# B&R Automation Studio project MappAssetInt (part 3)

#### ExportEventData.st
```iecst
// -------------------------------------------------------------------------------------------
// Read event data
// -------------------------------------------------------------------------------------------
FUNCTION_BLOCK ExportEventData
	// -------------------------------------------------------------------------------------------
	// Reset everything when enable is false
	IF NOT Enable THEN
		Status := ERR_FUB_ENABLE_FALSE;
		State := 0;
		RETURN;
	END_IF

	CASE State OF
		// -------------------------------------------------------------------------------------------
		// Wait for enable
		// -------------------------------------------------------------------------------------------
		0:
			IF Enable THEN

				// -------------------------------------------------------------------------------------------
				// Create file name
				RTC_gettime(ADR(RtcGettime));
				ExportType := ExportTypeJob;

				// Make sure we have data that can be exported
				IF RecordCount > 0 THEN
					Status := ERR_FUB_BUSY;
					CreateLoggerEntry(exASSETINT_LOG_INFO, ADR('start exporting data'), Logger);

					State := 1;
				ELSE

					CreateLoggerEntry(exASSETINT_LOG_INFO, ADR('no data to export'), Logger);
				END_IF
			END_IF

		// -------------------------------------------------------------------------------------------
		// Generate file name
		// -------------------------------------------------------------------------------------------
		1:
			// -------------------------------------------------------------------------------------------
			// Reset function blocks
			FileCreate_0.enable := FALSE;
			FileCreate_0();
			FileWrite_0.enable := FALSE;
			FileWrite_0();
			FileClose_0.enable := FALSE;
			FileClose_0();

			// -------------------------------------------------------------------------------------------
			// Export job data
			IF ExportType = ExportTypeJob THEN
				IF Configuration.JobStatistics THEN
					FileName := Configuration.JobStatisticsFileNamePattern;
				ELSE
					ExportType := ExportTypeShift;
				END_IF
			END_IF

			// -------------------------------------------------------------------------------------------
			// Export shift data
			IF ExportType = ExportTypeShift THEN
				IF Configuration.ShiftStatistics THEN
					FileName := Configuration.ShiftStatisticsFileNamePattern;
				ELSE
					ExportType := ExportTypeTimeline;
				END_IF
			END_IF

			// -------------------------------------------------------------------------------------------
			// Export timeline
			IF ExportType = ExportTypeTimeline THEN
				IF Configuration.JobStatistics THEN
					FileName := Configuration.TimelineFileNamePattern;
				ELSE
					State := 0;
					Status := ERR_OK;
					RETURN;
				END_IF
			END_IF

			// -------------------------------------------------------------------------------------------
			// Create date and time information
			ReplaceDateTime(ADR(FileName), ADR('%d'), RtcGettime.day);
			ReplaceDateTime(ADR(FileName), ADR('%m'), RtcGettime.month);
			ReplaceDateTime(ADR(FileName), ADR('%Y'), RtcGettime.year);

			ReplaceDateTime(ADR(FileName), ADR('%S'), RtcGettime.second);
			ReplaceDateTime(ADR(FileName), ADR('%M'), RtcGettime.month);
			ReplaceDateTime(ADR(FileName), ADR('%H'), RtcGettime.hour);

			idx := RecordCount - 1;
			Offset := 0;
			Status := ERR_FUB_BUSY;
			CreateLoggerEntry(exASSETINT_LOG_INFO, ADR('start exporting data'), Logger);

			State := 2;

		// -------------------------------------------------------------------------------------------
		// Delete old export file
		// -------------------------------------------------------------------------------------------
		2:
			FileDelete_0.enable := TRUE;
			FileDelete_0.pDevice := ADR(Device);
			FileDelete_0.pName := ADR(FileName);
			FileDelete_0();

			// -------------------------------------------------------------------------------------------
			// File delete successful
			IF FileDelete_0.status = ERR_OK  OR FileDelete_0.status = fiERR_FILE_NOT_FOUND THEN
				// Generate log entry
				TmpStr1 := 'delete old file ok > ';
				brsstrcat(ADR(TmpStr1), ADR(FileName));
				CreateLoggerEntry(exASSETINT_LOG_ALL, ADR(TmpStr1), Logger);

				State := 3;

			// Error
			ELSIF FileDelete_0.status <> ERR_FUB_BUSY THEN
				Status := FileDelete_0.status;
				State := 0;
			END_IF

		// -------------------------------------------------------------------------------------------
		// Create export file
		// -------------------------------------------------------------------------------------------
		3:
			FileCreate_0.enable := TRUE;
			FileCreate_0.pDevice := ADR(Device);
			FileCreate_0.pFile := ADR(FileName);
			FileCreate_0();

			// -------------------------------------------------------------------------------------------
			// File created successful
			IF FileCreate_0.status = ERR_OK THEN
				// Generate log entry
				TmpStr1 := 'create event file > ';
				brsstrcat(ADR(TmpStr1), ADR(FileName));
				CreateLoggerEntry(exASSETINT_LOG_ALL, ADR(TmpStr1), Logger);

				// Create header data depending on export file
				brsmemset(ADR(Buffer), 0, SIZEOF(Buffer));
				IF ExportType = ExportTypeJob THEN
					brsstrcat(ADR(Buffer), ADR(EXPORT_JOB_TITEL));
					brsstrcat(ADR(Buffer), ADR('$R'));
					brsstrcat(ADR(Buffer), ADR(EXPORT_JOB_HEADER));
					brsstrcat(ADR(Buffer), ADR('$R'));
				ELSIF ExportType = ExportTypeShift THEN
					brsstrcat(ADR(Buffer), ADR(EXPORT_SHIFT_TITEL));
					brsstrcat(ADR(Buffer), ADR('$R'));
					brsstrcat(ADR(Buffer), ADR(EXPORT_SHIFT_HEADER));
					brsstrcat(ADR(Buffer), ADR('$R'));
				ELSE
					brsstrcat(ADR(Buffer), ADR(EXPORT_TIMELINE_TITEL));
					brsstrcat(ADR(Buffer), ADR('$R'));
					brsstrcat(ADR(Buffer), ADR(EXPORT_TIMELINE_HEADER));
					brsstrcat(ADR(Buffer), ADR('$R'));
				END_IF

				State := 5;

			// Error
			ELSIF FileCreate_0.status <> ERR_FUB_BUSY THEN
				Status := FileCreate_0.status;
				State := 0;
			END_IF

		// -------------------------------------------------------------------------------------------
		// Generate data
		// -------------------------------------------------------------------------------------------
		4:
			// Reset buffer, copy new record
			brsmemset(ADR(Buffer), 0, SIZEOF(Buffer));
			brsmemcpy(ADR(RecordDataIntern), Memory + idx*SIZEOF(RecordDataIntern), SIZEOF(RecordDataIntern));

			// -------------------------------------------------------------------------------------------
			// Create row string for job and shift export
			IF (RecordDataIntern.EventType = RecordTypeJob AND ExportType = ExportTypeJob) OR (RecordDataIntern.EventType = RecordTypeShift AND ExportType = ExportTypeShift) THEN
				DT_TO_DTStructure(RecordDataIntern.TimeStart, ADR(DTStructure_0));
				TmpStr1 := Configuration.TimestampPattern;

				ReplaceDateTime(ADR(TmpStr1), ADR('%d'), DTStructure_0.day);
				ReplaceDateTime(ADR(TmpStr1), ADR('%m'), DTStructure_0.month);
				ReplaceDateTime(ADR(TmpStr1), ADR('%Y'), DTStructure_0.year);
				ReplaceDateTime(ADR(TmpStr1), ADR('%S'), DTStructure_0.second);
				ReplaceDateTime(ADR(TmpStr1), ADR('%M'), DTStructure_0.month);
				ReplaceDateTime(ADR(TmpStr1), ADR('%H'), DTStructure_0.hour);

				brsstrcat(ADR(Buffer), ADR(TmpStr1));
				brsstrcat(ADR(Buffer), ADR(Configuration.ColumnSeparator));

				DT_TO_DTStructure(RecordDataIntern.TimeEnd, ADR(DTStructure_0));
				TmpStr1 := Configuration.TimestampPattern;

				ReplaceDateTime(ADR(TmpStr1), ADR('%d'), DTStructure_0.day);
				ReplaceDateTime(ADR(TmpStr1), ADR('%m'), DTStructure_0.month);
				ReplaceDateTime(ADR(TmpStr1), ADR('%Y'), DTStructure_0.year);
				ReplaceDateTime(ADR(TmpStr1), ADR('%S'), DTStructure_0.second);
				ReplaceDateTime(ADR(TmpStr1), ADR('%M'), DTStructure_0.month);
				ReplaceDateTime(ADR(TmpStr1), ADR('%H'), DTStructure_0.hour);

				brsstrcat(ADR(Buffer), ADR(TmpStr1));
				brsstrcat(ADR(Buffer), ADR(Configuration.ColumnSeparator));

				brsstrcat(ADR(Buffer), ADR(RecordDataIntern.JobName));
				brsstrcat(ADR(Buffer), ADR(Configuration.ColumnSeparator));
				brsstrcat(ADR(Buffer), ADR(RecordDataIntern.CurrentUser));
				brsstrcat(ADR(Buffer), ADR(Configuration.ColumnSeparator));
				brsstrcat(ADR(Buffer), ADR(RecordDataIntern.AdditionalData));
				brsstrcat(ADR(Buffer), ADR(Configuration.ColumnSeparator));

				brsitoa(RecordDataIntern.TargetPieces, ADR(TmpStr1));
				brsstrcat(ADR(Buffer), ADR(TmpStr1));
				brsstrcat(ADR(Buffer), ADR(Configuration.ColumnSeparator));

				brsitoa(RecordDataIntern.GoodPieces, ADR(TmpStr1));
				brsstrcat(ADR(Buffer), ADR(TmpStr1));
				brsstrcat(ADR(Buffer), ADR(Configuration.ColumnSeparator));

				brsitoa(RecordDataIntern.RejectPieces, ADR(TmpStr1));
				brsstrcat(ADR(Buffer), ADR(TmpStr1));
				brsstrcat(ADR(Buffer), ADR(Configuration.ColumnSeparator));

				NormalizeFloat(RecordDataIntern.BadPieceRate, ADR(TmpStr1), Configuration);
				brsstrcat(ADR(Buffer), ADR(TmpStr1));
				brsstrcat(ADR(Buffer), ADR(Configuration.ColumnSeparator));

				lrealStr := NormalizeDateTime(RecordDataIntern.TotalTime.Hours);
				brsstrcat(ADR(Buffer), ADR(lrealStr));
				brsstrcat(ADR(Buffer), ADR(':'));
				lrealStr := NormalizeDateTime(RecordDataIntern.TotalTime.Minutes);
				brsstrcat(ADR(Buffer), ADR(lrealStr));
				brsstrcat(ADR(Buffer), ADR(':'));
				lrealStr := NormalizeDateTime(RecordDataIntern.TotalTime.Seconds);
				brsstrcat(ADR(Buffer), ADR(lrealStr));
				brsstrcat(ADR(Buffer), ADR(Configuration.ColumnSeparator));

				lrealStr := NormalizeDateTime(RecordDataIntern.ScheduledDowntime.Hours);
				brsstrcat(ADR(Buffer), ADR(lrealStr));
				brsstrcat(ADR(Buffer), ADR(':'));
				lrealStr := NormalizeDateTime(RecordDataIntern.ScheduledDowntime.Minutes);
				brsstrcat(ADR(Buffer), ADR(lrealStr));
				brsstrcat(ADR(Buffer), ADR(':'));
				lrealStr := NormalizeDateTime(RecordDataIntern.ScheduledDowntime.Seconds);
				brsstrcat(ADR(Buffer), ADR(lrealStr));
				brsstrcat(ADR(Buffer), ADR(Configuration.ColumnSeparator));

				lrealStr := NormalizeDateTime(RecordDataIntern.UnscheduledDowntime.Hours);
				brsstrcat(ADR(Buffer), ADR(lrealStr));
				brsstrcat(ADR(Buffer), ADR(':'));
				lrealStr := NormalizeDateTime(RecordDataIntern.UnscheduledDowntime.Minutes);
				brsstrcat(ADR(Buffer), ADR(lrealStr));
				brsstrcat(ADR(Buffer), ADR(':'));
				lrealStr := NormalizeDateTime(RecordDataIntern.UnscheduledDowntime.Seconds);
				brsstrcat(ADR(Buffer), ADR(lrealStr));
				brsstrcat(ADR(Buffer), ADR(Configuration.ColumnSeparator));

				lrealStr := NormalizeDateTime(RecordDataIntern.Uptime.Hours);
				brsstrcat(ADR(Buffer), ADR(lrealStr));
				brsstrcat(ADR(Buffer), ADR(':'));
				lrealStr := NormalizeDateTime(RecordDataIntern.Uptime.Minutes);
				brsstrcat(ADR(Buffer), ADR(lrealStr));
				brsstrcat(ADR(Buffer), ADR(':'));
				lrealStr := NormalizeDateTime(RecordDataIntern.Uptime.Seconds);
				brsstrcat(ADR(Buffer), ADR(lrealStr));
				brsstrcat(ADR(Buffer), ADR(Configuration.ColumnSeparator));

				lrealStr := NormalizeDateTime(RecordDataIntern.GoodProductionTime.Hours);
				brsstrcat(ADR(Buffer), ADR(lrealStr));
				brsstrcat(ADR(Buffer), ADR(':'));
				lrealStr := NormalizeDateTime(RecordDataIntern.GoodProductionTime.Minutes);
				brsstrcat(ADR(Buffer), ADR(lrealStr));
				brsstrcat(ADR(Buffer), ADR(':'));
				lrealStr := NormalizeDateTime(RecordDataIntern.GoodProductionTime.Seconds);
				brsstrcat(ADR(Buffer), ADR(lrealStr));
				brsstrcat(ADR(Buffer), ADR(Configuration.ColumnSeparator));

				lrealStr := NormalizeDateTime(RecordDataIntern.NominalProductionTime.Hours);
				brsstrcat(ADR(Buffer), ADR(lrealStr));
				brsstrcat(ADR(Buffer), ADR(':'));
				lrealStr := NormalizeDateTime(RecordDataIntern.NominalProductionTime.Minutes);
				brsstrcat(ADR(Buffer), ADR(lrealStr));
				brsstrcat(ADR(Buffer), ADR(':'));
				lrealStr := NormalizeDateTime(RecordDataIntern.NominalProductionTime.Seconds);
				brsstrcat(ADR(Buffer), ADR(lrealStr));
				brsstrcat(ADR(Buffer), ADR(Configuration.ColumnSeparator));

				NormalizeFloat(RecordDataIntern.NominalProductionTimeRate, ADR(TmpStr1), Configuration);
				brsstrcat(ADR(Buffer), ADR(TmpStr1));
				brsstrcat(ADR(Buffer), ADR(Configuration.ColumnSeparator));

				NormalizeFloat(RecordDataIntern.ScheduledDowntimeRate, ADR(TmpStr1), Configuration);
				brsstrcat(ADR(Buffer), ADR(TmpStr1));
				brsstrcat(ADR(Buffer), ADR(Configuration.ColumnSeparator));

				NormalizeFloat(RecordDataIntern.UnscheduledDowntimeRate, ADR(TmpStr1), Configuration);
				brsstrcat(ADR(Buffer), ADR(TmpStr1));
				brsstrcat(ADR(Buffer), ADR(Configuration.ColumnSeparator));

				NormalizeFloat(RecordDataIntern.CurrentProductionRate, ADR(TmpStr1), Configuration);
				brsstrcat(ADR(Buffer), ADR(TmpStr1));
				brsstrcat(ADR(Buffer), ADR(Configuration.ColumnSeparator));

				brsstrcat(ADR(Buffer), ADR(RecordDataIntern.ShiftName));
				brsstrcat(ADR(Buffer), ADR(Configuration.ColumnSeparator));
				brsstrcat(ADR(Buffer), ADR('$R'));

				State := 5;
			END_IF

			// -------------------------------------------------------------------------------------------
			// Export data for timeline

			IF (RecordDataIntern.EventType >= RecordTypeNoShift AND ExportType = ExportTypeTimeline) THEN
				// Create start time
				DT_TO_DTStructure(RecordDataIntern.TimeStart, ADR(DTStructure_0));
				TmpStr1 := Configuration.TimestampPattern;

				ReplaceDateTime(ADR(TmpStr1), ADR('%d'), DTStructure_0.day);
				ReplaceDateTime(ADR(TmpStr1), ADR('%m'), DTStructure_0.month);
				ReplaceDateTime(ADR(TmpStr1), ADR('%Y'), DTStructure_0.year);
				ReplaceDateTime(ADR(TmpStr1), ADR('%S'), DTStructure_0.second);
				ReplaceDateTime(ADR(TmpStr1), ADR('%M'), DTStructure_0.month);
				ReplaceDateTime(ADR(TmpStr1), ADR('%H'), DTStructure_0.hour);

				brsstrcat(ADR(Buffer), ADR(TmpStr1));
				brsstrcat(ADR(Buffer), ADR(Configuration.ColumnSeparator));

				// Add shift name
				brsstrcat(ADR(Buffer), ADR(RecordDataIntern.ShiftName));
				brsstrcat(ADR(Buffer), ADR(Configuration.ColumnSeparator));

				// Event is scheduled downtime
				IF RecordDataIntern.EventType = RecordTypeNoShift THEN
					brsstrcat(ADR(Buffer), ADR('No shift'));
				// Event is scheduled downtime
				ELSIF RecordDataIntern.EventType = RecordTypeDowntimeScheduled THEN
					brsstrcat(ADR(Buffer), ADR('Scheduled Downtime'));
				// Event is unscheduled downtime
				ELSIF RecordDataIntern.EventType = RecordTypeDowntimeUnscheduled THEN
					brsstrcat(ADR(Buffer), ADR('Unscheduled Downtime'));
				// Event is new shift
				ELSE
					brsstrcat(ADR(Buffer), ADR('Uptime'));
				END_IF
				brsstrcat(ADR(Buffer), ADR(Configuration.ColumnSeparator));

				// Additional data
				brsstrcat(ADR(Buffer), ADR(RecordDataIntern.AdditionalData));
				brsstrcat(ADR(Buffer), ADR(Configuration.ColumnSeparator));

				// Total time
				lrealStr := NormalizeDateTime(RecordDataIntern.TotalTime.Hours);
				brsstrcat(ADR(Buffer), ADR(lrealStr));
				brsstrcat(ADR(Buffer), ADR(':'));
				lrealStr := NormalizeDateTime(RecordDataIntern.TotalTime.Minutes);
				brsstrcat(ADR(Buffer), ADR(lrealStr));
				brsstrcat(ADR(Buffer), ADR(':'));
				lrealStr := NormalizeDateTime(RecordDataIntern.TotalTime.Seconds);
				brsstrcat(ADR(Buffer), ADR(lrealStr));
				brsstrcat(ADR(Buffer), ADR(Configuration.ColumnSeparator));

				// Job name
				brsstrcat(ADR(Buffer), ADR(RecordDataIntern.JobName));
				brsstrcat(ADR(Buffer), ADR(Configuration.ColumnSeparator));

				brsstrcat(ADR(Buffer), ADR('$R'));

				State := 5;
			END_IF

			// Increase counter
			IF idx = 0 THEN
				State := 6;
			ELSE
				idx := idx - 1;
			END_IF

		// -------------------------------------------------------------------------------------------
		// Write data
		// -------------------------------------------------------------------------------------------
		5:
			FileWrite_0.enable := TRUE;
			FileWrite_0.ident := FileCreate_0.ident;
			FileWrite_0.offset := Offset;
			FileWrite_0.pSrc := ADR(Buffer);
			FileWrite_0.len := brsstrlen(ADR(Buffer));
			FileWrite_0();

			// File created successful
			IF FileWrite_0.status = ERR_OK THEN
				// Generate log entry
				TmpStr1 := 'write idx ok > ';
				brsitoa(idx, ADR(TmpStr2));
				brsstrcat(ADR(TmpStr1), ADR(TmpStr2));
				CreateLoggerEntry(exASSETINT_LOG_ALL, ADR(TmpStr1), Logger);

				// Remember offset
				Offset := Offset + FileWrite_0.len;

				// Go to next step
				IF idx > 0 THEN
					State := 4;
				ELSE
					State := 6;
				END_IF

				// Error
			ELSIF FileWrite_0.status <> ERR_FUB_BUSY THEN
				Status := FileWrite_0.status;
				State := 0;
			END_IF

			// -------------------------------------------------------------------------------------------
			// Close file
			// -------------------------------------------------------------------------------------------
		6:
			FileClose_0.enable := TRUE;
			FileClose_0.ident := FileCreate_0.ident;
			FileClose_0();

			// File created successful
			IF FileClose_0.status = ERR_OK THEN
				// Generate log entry
				TmpStr1 := 'close export file ok > ';
				brsstrcat(ADR(TmpStr1), ADR(FileName));
				CreateLoggerEntry(exASSETINT_LOG_ALL, ADR(TmpStr1), Logger);

				// Proceed with shift export
				IF ExportType = ExportTypeJob THEN
					ExportType := ExportTypeShift;
					State := 1;
					// Proceed with timeline export
				ELSIF ExportType = ExportTypeShift THEN
					ExportType := ExportTypeTimeline;
					State := 1;
				ELSE
					// Finish up
					Status := ERR_OK;
					State := 0;
				END_IF

				// Error
			ELSIF FileClose_0.status <> ERR_FUB_BUSY THEN
				Status := FileClose_0.status;
				State := 0;
			END_IF
	END_CASE;

END_FUNCTION_BLOCK

// -------------------------------------------------------------------------------------------
// Format float according to configuration
// -------------------------------------------------------------------------------------------
FUNCTION NormalizeFloat
	brsftoa(value, ADR(tmpStr));
	idx := FindInstr(ADR(tmpStr), ADR('.')) + configuration.DecimalDigits + 1;
	IF idx >= brsstrlen(ADR(tmpStr)) THEN
		brsstrcpy(output, ADR(tmpStr));
	ELSE
		brsmemcpy(output, ADR(tmpStr), idx);
		brsmemset(output + idx, 0, 1);
	END_IF
	ReplaceString(output, ADR('.'), ADR(configuration.DecimalMark));
END_FUNCTION

// -------------------------------------------------------------------------------------------
// Add additional 0 when value is < 10
// -------------------------------------------------------------------------------------------
FUNCTION NormalizeDateTime
	IF(value < 10) THEN
		TmpStr1 := '0';
	ELSE
		TmpStr1 := '';
	END_IF
	brsitoa(value, ADR(TmpStr2));
	brsstrcat(ADR(TmpStr1), ADR(TmpStr2));

	brsmemcpy(ADR(NormalizeDateTime), ADR(TmpStr1), brsstrlen(ADR(TmpStr1)));

END_FUNCTION

// -------------------------------------------------------------------------------------------
// Find and replace date and time information
// -------------------------------------------------------------------------------------------
FUNCTION ReplaceDateTime
	lrealStr := NormalizeDateTime(value);
	ReplaceString(dataSTR, searchSTR, ADR(lrealStr));

	ReplaceDateTime := TRUE;
END_FUNCTION

// -------------------------------------------------------------------------------------------
// Find and replace string
// -------------------------------------------------------------------------------------------
FUNCTION ReplaceString
	IF (brsstrlen(dataSTR) >= brsstrlen(searchSTR)) THEN
		FOR idx:=0 TO brsstrlen(dataSTR) - brsstrlen(searchSTR) DO
			IF (brsmemcmp(dataSTR + idx, searchSTR, brsstrlen(searchSTR)) = 0) THEN
				// Move data around
				brsmemmove(dataSTR + idx + brsstrlen(replaceSTR), dataSTR + idx + brsstrlen(searchSTR), brsstrlen(dataSTR) - brsstrlen(searchSTR) + 1);
				brsmemcpy(dataSTR + idx, replaceSTR, brsstrlen(replaceSTR));
				// Set found flag and exit if only one hit is needed
				ReplaceString := TRUE;
				// Correct index for next search
				IF(brsstrlen(replaceSTR) > 0) THEN
					idx := idx + brsstrlen(replaceSTR);
				END_IF
				idx := idx - 1;
				// Exit if no data is left
				IF (brsstrlen(dataSTR) = 0 OR brsstrlen(dataSTR) < brsstrlen(searchSTR)) THEN
					EXIT;
				END_IF
			END_IF
		END_FOR;
	END_IF
END_FUNCTION
```

#### WriteConfiguration.st
```iecst
// -------------------------------------------------------------------------------------------
// Write configuration
// -------------------------------------------------------------------------------------------
FUNCTION_BLOCK WriteConfiguration
	// -------------------------------------------------------------------------------------------
	// Reset everything when enable is false
	IF NOT Enable THEN
		Status := ERR_FUB_ENABLE_FALSE;
		State := 0;
		RETURN;
	END_IF

	CASE State OF
		// -------------------------------------------------------------------------------------------
		// Wait for enable
		0:
			IF Enable THEN
				// Reset function blocks
				FileOpen_0.enable := FALSE;
				FileOpen_0();
				FileCreate_0.enable := FALSE;
				FileCreate_0();
				FileWrite_0.enable := FALSE;
				FileWrite_0();
				FileClose_0.enable := FALSE;
				FileClose_0();

				Status := ERR_FUB_BUSY;
				CreateLoggerEntry(exASSETINT_LOG_INFO, ADR('save configuration'), Logger);
				State := 1;
			END_IF

			// -------------------------------------------------------------------------------------------
			// Open file
		1:
			FileOpen_0.enable := TRUE;
			FileOpen_0.pDevice := ADR(Device);
			FileOpen_0.pFile := ADR('exAssetConfig');
			FileOpen_0.mode := fiREAD_WRITE;
			FileOpen_0();

			// File opened successful
			IF FileOpen_0.status = ERR_OK THEN
				// Generate log entry
				CreateLoggerEntry(exASSETINT_LOG_ALL, ADR('open configuration file ok'), Logger);

				// Remember ident go to next step
				Ident := FileOpen_0.ident;
				State := 3;

			// Create event file when it does not exist
			ELSIF FileOpen_0.status = fiERR_FILE_NOT_FOUND  THEN
				State := 2;

			// Error
			ELSIF FileOpen_0.status <> ERR_FUB_BUSY THEN
				Status := FileOpen_0.status;
				State := 0;
			END_IF

			// -------------------------------------------------------------------------------------------
			// Create file
		2:
			FileCreate_0.enable := TRUE;
			FileCreate_0.pDevice := ADR(Device);
			FileCreate_0.pFile := ADR('exAssetConfig');
			FileCreate_0();

			// File created successful
			IF FileCreate_0.status = ERR_OK THEN
				// Generate log entry
				CreateLoggerEntry(exASSETINT_LOG_ALL, ADR('created configuration file'), Logger);

				// Remember ident go to next step
				Ident := FileCreate_0.ident;
				State := 3;

				// Error
			ELSIF FileCreate_0.status <> ERR_FUB_BUSY THEN
				Status := FileCreate_0.status;
				State := 0;
			END_IF

			// -------------------------------------------------------------------------------------------
			// Write data
		3:
			FileWrite_0.enable := TRUE;
			FileWrite_0.ident := Ident;
			FileWrite_0.pSrc := ADR(Configuration);
			FileWrite_0.len := SIZEOF(Configuration);
			FileWrite_0();

			// File created successful
			IF FileWrite_0.status = ERR_OK THEN
				// Generate log entry
				CreateLoggerEntry(exASSETINT_LOG_ALL, ADR('write configuration file ok'), Logger);

				// Go to next step
				State := 4;

			// Error
			ELSIF FileWrite_0.status <> ERR_FUB_BUSY THEN
				Status := FileWrite_0.status;
				State := 0;
			END_IF

			// -------------------------------------------------------------------------------------------
			// Close file
		4:
			FileClose_0.enable := TRUE;
			FileClose_0.ident := Ident;
			FileClose_0();

			// File created successful
			IF FileClose_0.status = ERR_OK THEN
				// Generate log entry
				CreateLoggerEntry(exASSETINT_LOG_ALL, ADR('close configuration file ok'), Logger);

				// Finish up
				Status := ERR_OK;
				State := 0;

				// Error
			ELSIF FileClose_0.status <> ERR_FUB_BUSY THEN
				Status := FileClose_0.status;
				State := 0;
			END_IF
	END_CASE;

END_FUNCTION_BLOCK
```

#### ReadConfiguration.st
```iecst
// -------------------------------------------------------------------------------------------
// Read configuration
// -------------------------------------------------------------------------------------------
FUNCTION_BLOCK ReadConfiguration
	// -------------------------------------------------------------------------------------------
	// Reset everything when enable is false
	IF NOT Enable THEN
		Status := ERR_FUB_ENABLE_FALSE;
		State := 0;
		RETURN;
	END_IF

	CASE State OF
		// -------------------------------------------------------------------------------------------
		// Wait for enable
		0:
			IF Enable THEN
				// Reset function blocks
				FileOpen_0.enable := FALSE;
				FileOpen_0();
				FileRead_0.enable := FALSE;
				FileRead_0();
				FileClose_0.enable := FALSE;
				FileClose_0();

				Status := ERR_FUB_BUSY;
				CreateLoggerEntry(exASSETINT_LOG_INFO, ADR('reading configuration'), Logger);
				State := 1;
			END_IF

		// -------------------------------------------------------------------------------------------
		// Open event file
		1:
			// Open file
			FileOpen_0.enable := TRUE;
			FileOpen_0.pDevice := ADR(Device);
			FileOpen_0.pFile := ADR('exAssetConfig');
			FileOpen_0.mode := fiREAD_ONLY;
			FileOpen_0();

			// File opened successful
			IF FileOpen_0.status = ERR_OK THEN
				// Generate log entry
				CreateLoggerEntry(exASSETINT_LOG_ALL, ADR('opened event configuration'), Logger);

				// Go to next step
				State := 5;

			// Error
			ELSIF FileOpen_0.status <> ERR_FUB_BUSY THEN
				Status := FileOpen_0.status;
				State := 0;
			END_IF

		// -------------------------------------------------------------------------------------------
		// Read configuration data
		5:
			FileRead_0.enable := TRUE;
			FileRead_0.ident := FileOpen_0.ident;
			FileRead_0.pDest := ADR(Configuration);
			FileRead_0.len := FileOpen_0.filelen;
			FileRead_0();

			// File read successful
			IF FileRead_0.status = ERR_OK THEN
				// Generate log entry
				CreateLoggerEntry(exASSETINT_LOG_ALL, ADR('read event configuration'), Logger);

				State := 6;

			// Error
			ELSIF FileRead_0.status <> ERR_FUB_BUSY THEN
				Status := FileRead_0.status;
				State := 0;
			END_IF

		// -------------------------------------------------------------------------------------------
		// Close file
		6:
			FileClose_0.enable := TRUE;
			FileClose_0.ident := FileOpen_0.ident;
			FileClose_0();

			// File closed successful
			IF FileClose_0.status = ERR_OK THEN
				// Generate log entry
				CreateLoggerEntry(exASSETINT_LOG_ALL, ADR('closed event configuration'), Logger);

				// Go to next step
				Status := ERR_OK;
				State := 0;

				// Error
			ELSIF FileClose_0.status <> ERR_FUB_BUSY THEN
				Status := FileClose_0.status;
				State := 0;
			END_IF
	END_CASE;

END_FUNCTION_BLOCK
```

#### ReadLinkData.st
```iecst
// -------------------------------------------------------------------------------------------
// File version 1001
// -------------------------------------------------------------------------------------------
// Read configuration
// -------------------------------------------------------------------------------------------
FUNCTION_BLOCK ReadLinkData
	// -------------------------------------------------------------------------------------------
	// Reset everything when enable is false
	IF NOT Enable THEN
		Status := ERR_FUB_ENABLE_FALSE;
		State := 0;
		RETURN;
	END_IF

	CASE State OF
		// -------------------------------------------------------------------------------------------
		// Wait for enable
		0:
			IF Enable THEN
				// Reset function blocks
				FileOpen_0.enable := FALSE;
				FileOpen_0();
				FileRead_0.enable := FALSE;
				FileRead_0();
				FileClose_0.enable := FALSE;
				FileClose_0();

				Status := ERR_FUB_BUSY;
				CreateLoggerEntry(exASSETINT_LOG_INFO, ADR('reading link data'), Logger);
				State := 1;
			END_IF

		// -------------------------------------------------------------------------------------------
		// Open event file
		1:
			// Open file
			FileOpen_0.enable := TRUE;
			FileOpen_0.pDevice := ADR(Device);
			FileOpen_0.pFile := ADR('exAssetLink');
			FileOpen_0.mode := fiREAD_ONLY;
			FileOpen_0();

			// File opened successful
			IF FileOpen_0.status = ERR_OK THEN
				// Make sure backup data has correct size
				IF FileOpen_0.filelen <> SIZEOF(LinkRead) THEN
					CreateLoggerEntry(exASSETINT_LOG_ERROR, ADR('link backup data size is incorrect'), Logger);
					StatusRead := ERR_ASSET_LINK_SIZE;

					State := 6;
				ELSE
					CreateLoggerEntry(exASSETINT_LOG_ALL, ADR('open link data ok'), Logger);
					State := 5;
				END_IF

				// Error
			ELSIF FileOpen_0.status <> ERR_FUB_BUSY THEN
				Status := FileOpen_0.status;
				State := 0;
			END_IF

		// -------------------------------------------------------------------------------------------
		// Read configuration data
		5:
			FileRead_0.enable := TRUE;
			FileRead_0.ident := FileOpen_0.ident;
			FileRead_0.pDest := ADR(LinkRead);
			FileRead_0.len := FileOpen_0.filelen;
			FileRead_0();

			// File read successful
			IF FileRead_0.status = ERR_OK THEN
				// Make sure backup version is correct
				IF LinkRead.Version <> EXLINK_VERSION THEN
					CreateLoggerEntry(exASSETINT_LOG_ERROR, ADR('link backup data version is incorrect'), Logger);
					StatusRead := ERR_ASSET_LINK_VERSION;

				ELSE
					brsmemcpy(ADR(Link), ADR(LinkRead), SIZEOF(LinkRead));
					CreateLoggerEntry(exASSETINT_LOG_ALL, ADR('open link data ok'), Logger);
				END_IF

				State := 6;

			// Error
			ELSIF FileRead_0.status <> ERR_FUB_BUSY THEN
				Status := FileRead_0.status;
				State := 0;
			END_IF

		// -------------------------------------------------------------------------------------------
		// Close file
		6:
			FileClose_0.enable := TRUE;
			FileClose_0.ident := FileOpen_0.ident;
			FileClose_0();

			// File closed successful
			IF FileClose_0.status = ERR_OK THEN
				// Auto delete corrupt file
				IF StatusRead <> 0 THEN
					State := 7;
				ELSE
					// Generate log entry
					CreateLoggerEntry(exASSETINT_LOG_ALL, ADR('closed link data ok'), Logger);

					// Go to next step
					Status := ERR_OK;
					State := 0;
				END_IF

			// Error
			ELSIF FileClose_0.status <> ERR_FUB_BUSY THEN
				Status := FileClose_0.status;
				State := 0;
			END_IF

			// -------------------------------------------------------------------------------------------
			// Delete corrupt file
		7:
			FileDelete_0.enable := TRUE;
			FileDelete_0.pDevice := ADR(Device);
			FileDelete_0.pName := ADR('exAssetLink');
			FileDelete_0();

			// File delete successful
			IF FileDelete_0.status = ERR_OK THEN
				// Generate log entry
				CreateLoggerEntry(exASSETINT_LOG_ALL, ADR('delete corrupt link backup file ok'), Logger);

				Status := StatusRead;
				State := 0;

				// Error
			ELSIF FileDelete_0.status <> ERR_FUB_BUSY THEN
				Status := FileDelete_0.status;
				State := 0;
			END_IF
	END_CASE;

END_FUNCTION_BLOCK
```

#### WriteLinkData.st
```iecst
// -------------------------------------------------------------------------------------------
// File version 1000
// -------------------------------------------------------------------------------------------
// Write configuration
// -------------------------------------------------------------------------------------------
FUNCTION_BLOCK WriteLinkData
	// -------------------------------------------------------------------------------------------
	// Reset everything when enable is false
	IF NOT Enable THEN
		Status := ERR_FUB_ENABLE_FALSE;
		State := 0;
		RETURN;
	END_IF

	CASE State OF
		// -------------------------------------------------------------------------------------------
		// Wait for enable
		0:
			IF Enable THEN
				// Reset function blocks
				FileOpen_0.enable := FALSE;
				FileOpen_0();
				FileCreate_0.enable := FALSE;
				FileCreate_0();
				FileWrite_0.enable := FALSE;
				FileWrite_0();
				FileClose_0.enable := FALSE;
				FileClose_0();

				Status := ERR_FUB_BUSY;
				CreateLoggerEntry(exASSETINT_LOG_INFO, ADR('saving link data'), Logger);
				State := 1;
			END_IF

			// -------------------------------------------------------------------------------------------
			// Open file
		1:
			FileOpen_0.enable := TRUE;
			FileOpen_0.pDevice := ADR(Device);
			FileOpen_0.pFile := ADR('exAssetLink');
			FileOpen_0.mode := fiREAD_WRITE;
			FileOpen_0();

			// File opened successful
			IF FileOpen_0.status = ERR_OK THEN
				// Generate log entry
				CreateLoggerEntry(exASSETINT_LOG_ALL, ADR('open link data ok'), Logger);

				// Remember ident go to next step
				Ident := FileOpen_0.ident;
				State := 3;

			// Create event file when it does not exist
			ELSIF FileOpen_0.status = fiERR_FILE_NOT_FOUND  THEN
				State := 2;

			// Error
			ELSIF FileOpen_0.status <> ERR_FUB_BUSY THEN
				Status := FileOpen_0.status;
				State := 0;
			END_IF

			// -------------------------------------------------------------------------------------------
			// Create file
		2:
			FileCreate_0.enable := TRUE;
			FileCreate_0.pDevice := ADR(Device);
			FileCreate_0.pFile := ADR('exAssetLink');
			FileCreate_0();

			// File created successful
			IF FileCreate_0.status = ERR_OK THEN
				// Generate log entry
				CreateLoggerEntry(exASSETINT_LOG_ALL, ADR('create link data file'), Logger);

				// Remember ident go to next step
				Ident := FileCreate_0.ident;
				State := 3;

				// Error
			ELSIF FileCreate_0.status <> ERR_FUB_BUSY THEN
				Status := FileCreate_0.status;
				State := 0;
			END_IF

			// -------------------------------------------------------------------------------------------
			// Write data
		3:
			FileWrite_0.enable := TRUE;
			FileWrite_0.ident := Ident;
			FileWrite_0.pSrc := ADR(Link);
			FileWrite_0.len := SIZEOF(Link);
			FileWrite_0();

			// File created successful
			IF FileWrite_0.status = ERR_OK THEN
				// Generate log entry
				CreateLoggerEntry(exASSETINT_LOG_ALL, ADR('write link data ok'), Logger);

				// Go to next step
				State := 4;

			// Error
			ELSIF FileWrite_0.status <> ERR_FUB_BUSY THEN
				Status := FileWrite_0.status;
				State := 0;
			END_IF

			// -------------------------------------------------------------------------------------------
			// Close file
		4:
			FileClose_0.enable := TRUE;
			FileClose_0.ident := Ident;
			FileClose_0();

			// File created successful
			IF FileClose_0.status = ERR_OK THEN
				// Generate log entry
				CreateLoggerEntry(exASSETINT_LOG_ALL, ADR('close link data ok'), Logger);

				// Finish up
				Status := ERR_OK;
				State := 0;

				// Error
			ELSIF FileClose_0.status <> ERR_FUB_BUSY THEN
				Status := FileClose_0.status;
				State := 0;
			END_IF
	END_CASE;

END_FUNCTION_BLOCK
```

#### CalcStats.st
```iecst
// -------------------------------------------------------------------------------------------
// File version 1002
// -------------------------------------------------------------------------------------------
// Calculate current job statistics
FUNCTION CalcStatsJob
	// -------------------------------------------------------------------------------------------
	// Calculate total time, remember total time in milliseconds for accuaracy but convert to seconds for local calculations
	exLink.JobTotalTime := exLink.JobTotalTime + DiffLastCall;
	JobTotalTime := LREAL_TO_UDINT(exLink.JobTotalTime/1000);

	exLink.JobStatistics.TotalTime.Hours := JobTotalTime/3600;
	exLink.JobStatistics.TotalTime.Minutes := UDINT_TO_USINT((JobTotalTime - exLink.JobStatistics.TotalTime.Hours*3600)/60);
	exLink.JobStatistics.TotalTime.Seconds := UDINT_TO_USINT(JobTotalTime - exLink.JobStatistics.TotalTime.Hours*3600 - exLink.JobStatistics.TotalTime.Minutes*60);

	// Calculate scheduled downtime
	IF Downtime = exASSETINT_SCHEDULED_DOWNTIME THEN
		exLink.JobDowntimeScheduled := exLink.JobDowntimeScheduled + DiffLastCall;
		exLink.JobStatistics.ScheduledDowntime.Hours := exLink.JobDowntimeScheduled/3600000;
		exLink.JobStatistics.ScheduledDowntime.Minutes := UDINT_TO_USINT((exLink.JobDowntimeScheduled - exLink.JobStatistics.ScheduledDowntime.Hours*3600000)/60000);
		exLink.JobStatistics.ScheduledDowntime.Seconds := UDINT_TO_USINT((exLink.JobDowntimeScheduled - exLink.JobStatistics.ScheduledDowntime.Hours*3600000 - exLink.JobStatistics.ScheduledDowntime.Minutes*60000)/1000);
	END_IF

	// Calculate unscheduled downtime
	IF Downtime = exASSETINT_UNSCHEDULED_DOWNTIME THEN
		exLink.JobDowntimeUnscheduled := exLink.JobDowntimeUnscheduled + DiffLastCall;
		exLink.JobStatistics.UnscheduledDowntime.Hours := exLink.JobDowntimeUnscheduled/3600000;
		exLink.JobStatistics.UnscheduledDowntime.Minutes := UDINT_TO_USINT((exLink.JobDowntimeUnscheduled - exLink.JobStatistics.UnscheduledDowntime.Hours*3600000)/60000);
		exLink.JobStatistics.UnscheduledDowntime.Seconds := UDINT_TO_USINT((exLink.JobDowntimeUnscheduled - exLink.JobStatistics.UnscheduledDowntime.Hours*3600000 - exLink.JobStatistics.UnscheduledDowntime.Minutes*60000)/1000);
	END_IF

	// Calculate uptime
	IF Downtime = exASSETINT_NO_DOWNTIME THEN
		Uptime := JobTotalTime - exLink.JobDowntimeScheduled/1000 - exLink.JobDowntimeUnscheduled/1000;
		exLink.JobStatistics.Uptime.Hours := Uptime/3600;
		exLink.JobStatistics.Uptime.Minutes := UDINT_TO_USINT((Uptime - exLink.JobStatistics.Uptime.Hours*3600)/60);
		exLink.JobStatistics.Uptime.Seconds := UDINT_TO_USINT(Uptime - exLink.JobStatistics.Uptime.Hours*3600 - exLink.JobStatistics.Uptime.Minutes*60);
	END_IF

	// -------------------------------------------------------------------------------------------
	// Calculate counters
	IF exLink.JobStatistics.TotalPieces > exLink.JobStatistics.RejectPieces THEN
		exLink.JobStatistics.GoodPieces := exLink.JobStatistics.TotalPieces - exLink.JobStatistics.RejectPieces;
	ELSE
		exLink.JobStatistics.GoodPieces := 0;
		exLink.JobStatistics.RejectPieces := exLink.JobStatistics.TotalPieces;
	END_IF
	IF exLink.JobStatistics.TotalPieces > 0 THEN
		exLink.JobStatistics.BadPieceRate := UDINT_TO_REAL(exLink.JobStatistics.RejectPieces)/UDINT_TO_REAL(exLink.JobStatistics.TotalPieces);
	END_IF

	// -------------------------------------------------------------------------------------------
	// Additional times and rates
	NominalProductionTime := REAL_TO_UDINT(UDINT_TO_REAL(exLink.JobStatistics.TotalPieces)*(3600/Parameter.NominalProductionRate));
	exLink.JobStatistics.NominalProductionTime.Hours := NominalProductionTime/3600;
	exLink.JobStatistics.NominalProductionTime.Minutes := UDINT_TO_USINT((NominalProductionTime - exLink.JobStatistics.NominalProductionTime.Hours*3600)/60);
	exLink.JobStatistics.NominalProductionTime.Seconds := UDINT_TO_USINT(NominalProductionTime - exLink.JobStatistics.NominalProductionTime.Hours*3600 - exLink.JobStatistics.NominalProductionTime.Minutes*60);

	GoodProductionTime := REAL_TO_UDINT(UDINT_TO_REAL(exLink.JobStatistics.GoodPieces)*(3600/Parameter.NominalProductionRate));
	exLink.JobStatistics.GoodProductionTime.Hours := GoodProductionTime/3600;
	exLink.JobStatistics.GoodProductionTime.Minutes := UDINT_TO_USINT((GoodProductionTime - exLink.JobStatistics.GoodProductionTime.Hours*3600)/60);
	exLink.JobStatistics.GoodProductionTime.Seconds := UDINT_TO_USINT(GoodProductionTime - exLink.JobStatistics.GoodProductionTime.Hours*3600 - exLink.JobStatistics.GoodProductionTime.Minutes*60);

	IF exLink.JobDowntimeScheduled > 0 AND JobTotalTime > 0 THEN
		exLink.JobStatistics.ScheduledDowntimeRate := UDINT_TO_REAL(exLink.JobDowntimeScheduled/JobTotalTime)/1000;
	END_IF
	IF exLink.JobDowntimeUnscheduled > 0 AND JobTotalTime > 0 THEN
		exLink.JobStatistics.UnscheduledDowntimeRate := UDINT_TO_REAL(exLink.JobDowntimeUnscheduled/JobTotalTime)/1000;
	END_IF
	IF Uptime > 0 THEN
		exLink.JobStatistics.NominalProductionTimeRate := UDINT_TO_REAL(NominalProductionTime)/UDINT_TO_REAL(Uptime);
	END_IF
	IF JobTotalTime > 0 THEN
		exLink.JobStatistics.CurrentProductionRate := UDINT_TO_REAL(exLink.JobStatistics.TotalPieces)/UDINT_TO_REAL(JobTotalTime)*3600;
	END_IF

	brsmemcpy(ADR(JobStatistics), ADR(exLink.JobStatistics), SIZEOF(exLink.JobStatistics));
	CalcStatsJob := TRUE;
END_FUNCTION

// -------------------------------------------------------------------------------------------
// Calculate current shift statistics
FUNCTION CalcStatsShift
	// -------------------------------------------------------------------------------------------
	// Calculate total time, remember total time in milliseconds for accuaracy but convert to seconds for local calculations
	exLink.ShiftTotalTime := exLink.ShiftTotalTime + DiffLastCall;
	ShiftTotalTime := LREAL_TO_UDINT(exLink.ShiftTotalTime/1000);

	exLink.ShiftStatistics.TotalTime.Hours := ShiftTotalTime/3600;
	exLink.ShiftStatistics.TotalTime.Minutes := UDINT_TO_USINT((ShiftTotalTime - exLink.ShiftStatistics.TotalTime.Hours*3600)/60);
	exLink.ShiftStatistics.TotalTime.Seconds := UDINT_TO_USINT(ShiftTotalTime - exLink.ShiftStatistics.TotalTime.Hours*3600 - exLink.ShiftStatistics.TotalTime.Minutes*60);

	// Calculate scheduled downtime
	IF Downtime = exASSETINT_SCHEDULED_DOWNTIME THEN
		exLink.ShiftDowntimeScheduled := exLink.ShiftDowntimeScheduled + DiffLastCall;
		exLink.ShiftStatistics.ScheduledDowntime.Hours := exLink.ShiftDowntimeScheduled/3600000;
		exLink.ShiftStatistics.ScheduledDowntime.Minutes := UDINT_TO_USINT((exLink.ShiftDowntimeScheduled - exLink.ShiftStatistics.ScheduledDowntime.Hours*3600000)/60000);
		exLink.ShiftStatistics.ScheduledDowntime.Seconds := UDINT_TO_USINT((exLink.ShiftDowntimeScheduled - exLink.ShiftStatistics.ScheduledDowntime.Hours*3600000 - exLink.ShiftStatistics.ScheduledDowntime.Minutes*60000)/1000);
	END_IF

	// Calculate scheduled downtime
	IF Downtime = exASSETINT_UNSCHEDULED_DOWNTIME THEN
		exLink.ShiftDowntimeUnscheduled := exLink.ShiftDowntimeUnscheduled + DiffLastCall;
		exLink.ShiftStatistics.UnscheduledDowntime.Hours := exLink.ShiftDowntimeUnscheduled/3600000;
		exLink.ShiftStatistics.UnscheduledDowntime.Minutes := UDINT_TO_USINT((exLink.ShiftDowntimeUnscheduled - exLink.ShiftStatistics.UnscheduledDowntime.Hours*3600000)/60000);
		exLink.ShiftStatistics.UnscheduledDowntime.Seconds := UDINT_TO_USINT((exLink.ShiftDowntimeUnscheduled - exLink.ShiftStatistics.UnscheduledDowntime.Hours*3600000 - exLink.ShiftStatistics.UnscheduledDowntime.Minutes*60000)/1000);
	END_IF

	// Calculate uptime
	IF Downtime = exASSETINT_NO_DOWNTIME THEN
		Uptime := ShiftTotalTime - exLink.ShiftDowntimeScheduled/1000 - exLink.ShiftDowntimeUnscheduled/1000;
		exLink.ShiftStatistics.Uptime.Hours := Uptime/3600;
		exLink.ShiftStatistics.Uptime.Minutes := UDINT_TO_USINT((Uptime - exLink.ShiftStatistics.Uptime.Hours*3600)/60);
		exLink.ShiftStatistics.Uptime.Seconds := UDINT_TO_USINT(Uptime - exLink.ShiftStatistics.Uptime.Hours*3600 - exLink.ShiftStatistics.Uptime.Minutes*60);
	END_IF

	// -------------------------------------------------------------------------------------------
	// Calculate counters
	exLink.ShiftStatistics.TargetPieces := LREAL_TO_UDINT(UDINT_TO_REAL(ShiftTotalTime)/3600*Parameter.NominalProductionRate);
	IF exLink.ShiftStatistics.TotalPieces > exLink.ShiftStatistics.RejectPieces THEN
		exLink.ShiftStatistics.GoodPieces := exLink.ShiftStatistics.TotalPieces - exLink.ShiftStatistics.RejectPieces;
	ELSE
		exLink.ShiftStatistics.GoodPieces := 0;
		exLink.ShiftStatistics.RejectPieces := exLink.ShiftStatistics.TotalPieces;
	END_IF
	IF exLink.ShiftStatistics.TotalPieces > 0 THEN
		exLink.ShiftStatistics.BadPieceRate := UDINT_TO_REAL(exLink.ShiftStatistics.RejectPieces)/UDINT_TO_REAL(exLink.ShiftStatistics.TotalPieces);
	END_IF

	// -------------------------------------------------------------------------------------------
	// Additional times and rates
	NominalProductionTime := REAL_TO_UDINT(UDINT_TO_REAL(exLink.ShiftStatistics.TotalPieces)*(3600/Parameter.NominalProductionRate));
	exLink.ShiftStatistics.NominalProductionTime.Hours := NominalProductionTime/3600;
	exLink.ShiftStatistics.NominalProductionTime.Minutes := UDINT_TO_USINT((NominalProductionTime - exLink.ShiftStatistics.NominalProductionTime.Hours*3600)/60);
	exLink.ShiftStatistics.NominalProductionTime.Seconds := UDINT_TO_USINT(NominalProductionTime - exLink.ShiftStatistics.NominalProductionTime.Hours*3600 - exLink.ShiftStatistics.NominalProductionTime.Minutes*60);

	GoodProductionTime := REAL_TO_UDINT(UDINT_TO_REAL(exLink.ShiftStatistics.GoodPieces)*(3600/Parameter.NominalProductionRate));
	exLink.ShiftStatistics.GoodProductionTime.Hours := GoodProductionTime/3600;
	exLink.ShiftStatistics.GoodProductionTime.Minutes := UDINT_TO_USINT((GoodProductionTime - exLink.ShiftStatistics.GoodProductionTime.Hours*3600)/60);
	exLink.ShiftStatistics.GoodProductionTime.Seconds := UDINT_TO_USINT(GoodProductionTime - exLink.ShiftStatistics.GoodProductionTime.Hours*3600 - exLink.ShiftStatistics.GoodProductionTime.Minutes*60);

	IF exLink.ShiftDowntimeScheduled > 0 AND ShiftTotalTime > 0 THEN
		exLink.ShiftStatistics.ScheduledDowntimeRate := UDINT_TO_REAL(exLink.ShiftDowntimeScheduled/ShiftTotalTime)/1000;
	END_IF
	IF exLink.ShiftDowntimeUnscheduled > 0 AND ShiftTotalTime > 0 THEN
		exLink.ShiftStatistics.UnscheduledDowntimeRate := UDINT_TO_REAL(exLink.ShiftDowntimeUnscheduled/ShiftTotalTime)/1000;
	END_IF
	IF Uptime > 0 THEN
		exLink.ShiftStatistics.NominalProductionTimeRate := UDINT_TO_REAL(NominalProductionTime)/UDINT_TO_REAL(Uptime);
	END_IF
	IF ShiftTotalTime > 0 THEN
		exLink.ShiftStatistics.CurrentProductionRate := UDINT_TO_REAL(exLink.ShiftStatistics.TotalPieces)/UDINT_TO_REAL(ShiftTotalTime)*3600;
	END_IF

	brsmemcpy(ADR(ShiftStatistics), ADR(exLink.ShiftStatistics), SIZEOF(exLink.ShiftStatistics));
	CalcStatsShift := TRUE;
END_FUNCTION
```

#### TrackShift.st
```iecst
// -------------------------------------------------------------------------------------------
// File version 1001
// -------------------------------------------------------------------------------------------

// -------------------------------------------------------------------------------------------
// Handle shift change
FUNCTION TrackShiftChange
	// -------------------------------------------------------------------------------------------
	// Handle shift change over days
	IF Internal.PowerOffTime <> DT#1970-01-01-00:00:00 THEN
		DiffTime := DiffDT(Internal.CurrentTime.DT1, Internal.PowerOffTime);
		DiffTime := DiffTime - exLink.ShiftSecondsToEnd;
	END_IF

	// -------------------------------------------------------------------------------------------
	// Track current shift
	Internal.ShiftName := '';
	Internal.ShiftId := -1;
	FOR Internal.x := 0 TO SIZEOF(exLink.Configuration.Shifts)/SIZEOF(exLink.Configuration.Shifts[0]) - 1 DO
		// Shift ends on same day
		IF exLink.Configuration.Shifts[Internal.x].TotalTime.Start < exLink.Configuration.Shifts[Internal.x].TotalTime.End THEN
			IF Internal.TimeOfDay >= exLink.Configuration.Shifts[Internal.x].TotalTime.Start AND Internal.TimeOfDay <= exLink.Configuration.Shifts[Internal.x].TotalTime.End THEN
				Internal.ShiftName := exLink.Configuration.Shifts[Internal.x].Name;
				Internal.ShiftId := UINT_TO_SINT(Internal.x);
				exLink.ShiftSecondsToEnd := (TOD_TO_UDINT(exLink.Configuration.Shifts[Internal.x].TotalTime.End) - TOD_TO_UDINT(Internal.TimeOfDay))/1000;
				EXIT;
			END_IF
			// Shift ends next day
		ELSE
			IF Internal.TimeOfDay >= exLink.Configuration.Shifts[Internal.x].TotalTime.Start OR Internal.TimeOfDay <= exLink.Configuration.Shifts[Internal.x].TotalTime.End THEN
				Internal.ShiftName := exLink.Configuration.Shifts[Internal.x].Name;
				Internal.ShiftId := UINT_TO_SINT(Internal.x);
				IF Internal.TimeOfDay >= exLink.Configuration.Shifts[Internal.x].TotalTime.Start THEN
					exLink.ShiftSecondsToEnd := (TOD_TO_UDINT(TOD#23:59:59.999) - TOD_TO_UDINT(Internal.TimeOfDay) + TOD_TO_UDINT(exLink.Configuration.Shifts[Internal.x].TotalTime.End))/1000;
				ELSE
					exLink.ShiftSecondsToEnd := (TOD_TO_UDINT(exLink.Configuration.Shifts[Internal.x].TotalTime.End) - TOD_TO_UDINT(Internal.TimeOfDay))/1000;
				END_IF
				EXIT;
			END_IF
		END_IF
	END_FOR;

	// -------------------------------------------------------------------------------------------
	// Track current shift scheduled downtime
	IF exLink.ShiftId >= 0 THEN
		FOR Internal.x := 0 TO SIZEOF(exLink.Configuration.Shifts[exLink.ShiftId].ScheduledDowntime)/SIZEOF(exLink.Configuration.Shifts[exLink.ShiftId].ScheduledDowntime[0]) - 1 DO
			// Make sure we have a valid configuration
			IF TOD_TO_UDINT(exLink.Configuration.Shifts[exLink.ShiftId].ScheduledDowntime[Internal.x].Start) <> 0 OR TOD_TO_UDINT(exLink.Configuration.Shifts[exLink.ShiftId].ScheduledDowntime[Internal.x].End) <> 0 THEN
				// Downtime ends on same day
				IF exLink.Configuration.Shifts[exLink.ShiftId].ScheduledDowntime[Internal.x].Start < exLink.Configuration.Shifts[exLink.ShiftId].ScheduledDowntime[Internal.x].End THEN
					IF Internal.TimeOfDay >= exLink.Configuration.Shifts[exLink.ShiftId].ScheduledDowntime[Internal.x].Start AND Internal.TimeOfDay < exLink.Configuration.Shifts[exLink.ShiftId].ScheduledDowntime[Internal.x].End THEN
						Internal.Downtime := exASSETINT_SCHEDULED_DOWNTIME;
						Internal.DowntimeReason := exLink.Configuration.Shifts[exLink.ShiftId].ScheduledDowntime[Internal.x].Reason;
						EXIT;
					END_IF
				ELSE
					IF Internal.TimeOfDay >= exLink.Configuration.Shifts[exLink.ShiftId].ScheduledDowntime[Internal.x].Start OR Internal.TimeOfDay < exLink.Configuration.Shifts[exLink.ShiftId].ScheduledDowntime[Internal.x].End THEN
						Internal.Downtime := exASSETINT_SCHEDULED_DOWNTIME;
						Internal.DowntimeReason := exLink.Configuration.Shifts[exLink.ShiftId].ScheduledDowntime[Internal.x].Reason;
						EXIT;
					END_IF
				END_IF
			END_IF
		END_FOR;
	END_IF

	// -------------------------------------------------------------------------------------------
	// Handle shift change
	IF (exLink.ShiftStatistics.ShiftName <> Internal.ShiftName) OR (DiffTime > 0) THEN
		// Transfer stats to record, make sure structures are allignent
		brsmemset(ADR(Internal.RecordData), 0, SIZEOF(Internal.RecordData));

		IF Internal.ShiftName <> '' THEN
			Internal.TmpStr1 := 'new shift started ';
			brsstrcat(ADR(Internal.TmpStr1), ADR(Internal.ShiftName));
			CreateLoggerEntry(exASSETINT_LOG_INFO, ADR(Internal.TmpStr1), Logger);
		ELSIF exLink.ShiftStatistics.ShiftName <> '' THEN
			Internal.TmpStr1 := 'shift ended ';
			brsstrcat(ADR(Internal.TmpStr1), ADR(exLink.ShiftStatistics.ShiftName));
			CreateLoggerEntry(exASSETINT_LOG_INFO, ADR(Internal.TmpStr1), Logger);
		END_IF

		// Only store data when shift name was not empty
		IF exLink.ShiftStatistics.ShiftName <> '' THEN
			// Collect data for record
			Internal.RecordData.EventType := RecordTypeShift;
			Internal.RecordData.TimeStart := exLink.ShiftStatistics.StartTime;
			// Use power off time for shift end
			IF DiffTime > 0 THEN
				DT_TO_DTStructure(Internal.PowerOffTime, ADR(exLink.StatsLastCall));
			END_IF
			Internal.RecordData.TimeEnd := DTStructure_TO_DT(ADR(exLink.StatsLastCall));
			Internal.RecordData.CurrentUser := exLink.ShiftStatistics.CurrentUser;
			Internal.RecordData.AdditionalData := exLink.ShiftStatistics.AdditionalData;
			Internal.RecordData.ShiftName := exLink.ShiftStatistics.ShiftName;
			Internal.RecordData.JobName := exLink.JobStatistics.JobName;
			Internal.RecordData.TotalPieces := exLink.ShiftStatistics.TotalPieces;
			Internal.RecordData.GoodPieces := exLink.ShiftStatistics.GoodPieces;
			Internal.RecordData.RejectPieces := exLink.ShiftStatistics.RejectPieces;
			Internal.RecordData.BadPieceRate := exLink.ShiftStatistics.BadPieceRate;
			Internal.RecordData.TargetPieces := exLink.ShiftStatistics.TargetPieces;
			Internal.RecordData.TotalTime := exLink.ShiftStatistics.TotalTime;
			Internal.RecordData.ScheduledDowntime := exLink.ShiftStatistics.ScheduledDowntime;
			Internal.RecordData.UnscheduledDowntime := exLink.ShiftStatistics.UnscheduledDowntime;
			Internal.RecordData.Uptime := exLink.ShiftStatistics.Uptime;
			Internal.RecordData.GoodProductionTime := exLink.ShiftStatistics.GoodProductionTime;
			Internal.RecordData.NominalProductionTime := exLink.ShiftStatistics.NominalProductionTime;
			Internal.RecordData.NominalProductionTimeRate := exLink.ShiftStatistics.NominalProductionTimeRate;
			Internal.RecordData.UnscheduledDowntimeRate := exLink.ShiftStatistics.UnscheduledDowntimeRate;
			Internal.RecordData.CurrentProductionRate := exLink.ShiftStatistics.CurrentProductionRate;

			Internal.State := exASSETINT_STATE_STORE_EVENT;
			TrackShiftChange := TRUE;

		ELSE
			TrackShiftChange := FALSE;

		END_IF

		// Remember job start time
		IF exLink.JobStatistics.StartTime = DT#1970-01-01-00:00:00 THEN
			exLink.JobStatistics.StartTime := Internal.CurrentTime.DT1;
		END_IF

		// Reset stats
		brsmemset(ADR(Info.ShiftStatistics), 0, SIZEOF(Info.ShiftStatistics));
		brsmemset(ADR(exLink.ShiftStatistics), 0, SIZEOF(exLink.ShiftStatistics));

		exLink.ShiftTotalTime := 0;
		exLink.ShiftDowntimeScheduled := 0;
		exLink.ShiftDowntimeUnscheduled := 0;

		// Transfer data to shift stats
		exLink.ShiftId := Internal.ShiftId;
		exLink.ShiftStatistics.StartTime := Internal.CurrentTime.DT1;
		exLink.ShiftStatistics.ShiftName := Internal.ShiftName;
		exLink.ShiftStatistics.CurrentUser := Parameters.CurrentUser;
		exLink.ShiftStatistics.AdditionalData := Parameters.AdditionalData;
	END_IF

	Internal.PowerOffTime := DT#1970-01-01-00:00:00;
END_FUNCTION
```

#### TrackProduction.st
```iecst
// -------------------------------------------------------------------------------------------
// File version 1002
// -------------------------------------------------------------------------------------------

// -------------------------------------------------------------------------------------------
// Handle production state change
FUNCTION TrackProductionState
	IF (exLink.ShiftStatistics.ShiftName <> exLink.ProductionShiftName) OR (exLink.JobStatistics.JobName <> exLink.ProductionJobName AND exLink.ShiftId >= 0) OR (exLink.JobStatistics.CurrentUser <> exLink.ProductionUserName AND exLink.ShiftId >= 0) OR (Internal.Downtime <> exLink.ProductionDowntime AND exLink.ShiftId >= 0) OR (Internal.DowntimeReason <> exLink.ProductionDowntimeReason AND exLink.ProductionDowntime > exASSETINT_NO_DOWNTIME) THEN

		// Transfer stats to record, make sure structures are allignent
		brsmemset(ADR(Internal.RecordData), 0, SIZEOF(Internal.RecordData));

		// Collect data for record
		Internal.RecordData.TimeStart := exLink.ProductionStateStart;
		Internal.RecordData.TimeEnd := Internal.CurrentTime.DT1;
		Internal.RecordData.ShiftName := exLink.ProductionShiftName;
		Internal.RecordData.JobName := exLink.ProductionJobName;

		Internal.ProductionTotalTime := LREAL_TO_UDINT(exLink.ProductionTotalTime/1000);
		Internal.RecordData.TotalTime.Hours := Internal.ProductionTotalTime/3600;
		Internal.RecordData.TotalTime.Minutes := UDINT_TO_USINT((Internal.ProductionTotalTime - Internal.RecordData.TotalTime.Hours*3600)/60);
		Internal.RecordData.TotalTime.Seconds := UDINT_TO_USINT(Internal.ProductionTotalTime - Internal.RecordData.TotalTime.Hours*3600 - Internal.RecordData.TotalTime.Minutes*60);

		// -------------------------------------------------------------------------------------------
		// State change is shift
		IF exLink.ShiftStatistics.ShiftName <> exLink.ProductionShiftName THEN
			// Set event type
			Internal.RecordData.EventType := UDINT_TO_UINT(exLink.ProductionState + 2);

			// Create log message and production state
			Internal.TmpStr1 := 'shift changed from ';
			IF exLink.ProductionState = exASSETINT_STATE_NO_SHIFT_ACTIVE THEN
				brsstrcat(ADR(Internal.TmpStr1), ADR('no shift '));
			ELSE
				brsstrcat(ADR(Internal.TmpStr1), ADR(exLink.ProductionShiftName));
			END_IF
			brsstrcat(ADR(Internal.TmpStr1), ADR(' to '));

			// State change is to no shift
			IF exLink.ShiftStatistics.ShiftName = '' THEN
				brsstrcat(ADR(Internal.TmpStr1), ADR('no shift'));
				exLink.ProductionState := exASSETINT_STATE_NO_SHIFT_ACTIVE;

				// State change is to uptime
			ELSE
				brsstrcat(ADR(Internal.TmpStr1), ADR(exLink.ShiftStatistics.ShiftName));
				exLink.ProductionState := UDINT_TO_UINT(Internal.Downtime + 1);
			END_IF

			// Remember shift name
			exLink.ProductionShiftName := exLink.ShiftStatistics.ShiftName;

			// -------------------------------------------------------------------------------------------
			// State change is job
		ELSIF exLink.JobStatistics.JobName <> exLink.ProductionJobName THEN
			// Set event type
			Internal.RecordData.EventType := UDINT_TO_UINT(exLink.ProductionState + 2);

			// Create log message
			Internal.TmpStr1 := 'job changed from ';
			IF exLink.ProductionJobName = '' THEN
				brsstrcat(ADR(Internal.TmpStr1), ADR('none '));
			ELSE
				brsstrcat(ADR(Internal.TmpStr1), ADR(exLink.ProductionJobName));
			END_IF
			brsstrcat(ADR(Internal.TmpStr1), ADR(' to '));

			// Job name is empty
			IF exLink.JobStatistics.JobName = '' THEN
				brsstrcat(ADR(Internal.TmpStr1), ADR('none'));
				// State change is to uptime
			ELSE
				brsstrcat(ADR(Internal.TmpStr1), ADR(exLink.JobStatistics.JobName));
			END_IF

			// Remember job name
			exLink.ProductionJobName := exLink.JobStatistics.JobName;

			// ----------------------------------------------------
			// State change is new user
		ELSIF exLink.JobStatistics.CurrentUser <> exLink.ProductionUserName THEN
			// Set event type
			Internal.RecordData.EventType := RecordTypeUserChange;

			// Create log message
			Internal.TmpStr1 := 'user changed from ';
			IF exLink.ProductionUserName <> '' THEN
				brsstrcat(ADR(Internal.TmpStr1), ADR(exLink.ProductionUserName));
			ELSE
				brsstrcat(ADR(Internal.TmpStr1), ADR('none'));
			END_IF
			brsstrcat(ADR(Internal.TmpStr1), ADR(' to '));

			// User name is empty
			IF Parameters.CurrentUser = '' THEN
				brsstrcat(ADR(Internal.TmpStr1), ADR('none'));
			ELSE
				brsstrcat(ADR(Internal.TmpStr1), ADR(Parameters.CurrentUser));
			END_IF

			// Remember use name
			exLink.ProductionUserName := exLink.JobStatistics.CurrentUser;
			Internal.RecordData.AdditionalData := LEFT(Internal.TmpStr1, SIZEOF(Internal.RecordData.AdditionalData));

			// ----------------------------------------------------
			// State change is downtime
		ELSIF Internal.Downtime <> exLink.ProductionDowntime THEN
			// Set event type
			Internal.RecordData.EventType := UDINT_TO_UINT(exLink.ProductionState + 2);

			// Create log message
			Internal.TmpStr1 := 'production state changed from ';
			IF exLink.ProductionState = exASSETINT_STATE_UPTIME THEN
				brsstrcat(ADR(Internal.TmpStr1), ADR('uptime to '));
			ELSIF exLink.ProductionState = exASSETINT_STATE_SCHDL_DOWNTIME THEN
				brsstrcat(ADR(Internal.TmpStr1), ADR('scheduled dt to '));
			ELSE
				brsstrcat(ADR(Internal.TmpStr1), ADR('unscheduled dt to '));
			END_IF

			IF Internal.Downtime = exASSETINT_NO_DOWNTIME THEN
				brsstrcat(ADR(Internal.TmpStr1), ADR('no downtime'));
			ELSIF Internal.Downtime = exASSETINT_SCHEDULED_DOWNTIME THEN
				brsstrcat(ADR(Internal.TmpStr1), ADR('scheduled dt > '));
				brsstrcat(ADR(Internal.TmpStr1), ADR(Internal.DowntimeReason));
			ELSE
				brsstrcat(ADR(Internal.TmpStr1), ADR('unscheduled dt > '));
				brsstrcat(ADR(Internal.TmpStr1), ADR(Internal.DowntimeReason));
			END_IF

			IF exLink.ProductionState = exASSETINT_STATE_SCHDL_DOWNTIME OR exLink.ProductionState = exASSETINT_STATE_UNSCH_DOWNTIME THEN
				Internal.RecordData.AdditionalData := exLink.ProductionDowntimeReason;
			END_IF

			// Remember downtime and reason, set production state
			exLink.ProductionDowntime := Internal.Downtime;
			exLink.ProductionDowntimeReason := Internal.DowntimeReason;
			exLink.ProductionState := UDINT_TO_UINT(Internal.Downtime + 1);

			// ----------------------------------------------------
			// State change is downtime reason
		ELSE
			// Set event type
			Internal.RecordData.EventType := UDINT_TO_UINT(exLink.ProductionState + 2);

			// Create log message
			Internal.TmpStr1 := 'dt reason changed from ';
			IF exLink.ProductionDowntimeReason <> '' THEN
				brsstrcat(ADR(Internal.TmpStr1), ADR(exLink.ProductionDowntimeReason));
			ELSE
				brsstrcat(ADR(Internal.TmpStr1), ADR('none'));
			END_IF
			brsstrcat(ADR(Internal.TmpStr1), ADR(' to '));
			IF Internal.DowntimeReason <> '' THEN
				brsstrcat(ADR(Internal.TmpStr1), ADR(Internal.DowntimeReason));
			ELSE
				brsstrcat(ADR(Internal.TmpStr1), ADR('none'));
			END_IF

			Internal.RecordData.AdditionalData := exLink.ProductionDowntimeReason;

			// Remember downtime reason
			exLink.ProductionDowntimeReason := Internal.DowntimeReason;
		END_IF

		CreateLoggerEntry(exASSETINT_LOG_INFO, ADR(Internal.TmpStr1), Logger);

		// Remember production start
		IF exLink.ProductionStateStart <> DT#1970-01-01-00:00:00 THEN
			exLink.ProductionStateStart := Internal.CurrentTime.DT1;
			exLink.ProductionTotalTime := 0;

			// Create new event
			Internal.State := exASSETINT_STATE_STORE_EVENT;

			// Just remember start time after cold start
		ELSE
			exLink.ProductionStateStart := Internal.CurrentTime.DT1;
		END_IF
		TrackProductionState := TRUE;

	ELSE
		TrackProductionState := FALSE;

	END_IF

	// Remember production duration
	IF Internal.StatsRefresh.Q THEN
		// Get time difference between calls
		Internal.DiffLastCallProduction := DiffT(clock_ms(), Internal.TimeLastCallProduction);
		Internal.TimeLastCallProduction := clock_ms();
		IF Internal.DiffLastCallProduction = 16#FFFFFFFF THEN
			CreateLoggerEntry(exASSETINT_LOG_INFO, ADR('diff timer overflow'), Logger);
		ELSE
			exLink.ProductionTotalTime := exLink.ProductionTotalTime + Internal.DiffLastCallProduction;
		END_IF
	END_IF

END_FUNCTION
```

#### common.st
```iecst
// -------------------------------------------------------------------------------------------
// Go to error state
FUNCTION CreateErrorState
	Internal.StateError := Internal.State;
	Internal.State := exASSETINT_STATE_ERROR;
	CreateErrorState := ErrorID;
END_FUNCTION

// -------------------------------------------------------------------------------------------
// Handle log buffer
FUNCTION CreateLoggerEntry
	// Make sure we dont flood Logger
	IF LogMsg <> LastMsg AND LogLevel <= LOG_LEVEL THEN
		// Make sure log message fits
		IF brsstrlen(ADR(LogMsg)) > LOG_LEN THEN
			LogMsg := '*** log meassage exceeds maximum length ***';
		END_IF
		// Move ring buffer around
		brsmemmove(LogBuffer+LOG_LEN+1, LogBuffer, LOG_LEN*(LOG_NUM-1));
		brsstrcpy(LogBuffer, ADR(''));
		// Create time information
		RTC_gettime(ADR(RtcGettime));
		IF(RtcGettime.day < 10) THEN
			brsstrcat(LogBuffer, ADR('0'));
		END_IF
		brsitoa(RtcGettime.day, ADR(TmpStr));
		brsstrcat(LogBuffer, ADR(TmpStr));
		brsitoa(RtcGettime.day, ADR(TmpStr));
		brsstrcat(LogBuffer, ADR('.'));
		IF(RtcGettime.month < 10) THEN
			brsstrcat(LogBuffer, ADR('0'));
		END_IF
		brsitoa(RtcGettime.month, ADR(TmpStr));
		brsstrcat(LogBuffer, ADR(TmpStr));
		brsstrcat(LogBuffer, ADR(' '));
		IF(RtcGettime.hour < 10) THEN
			brsstrcat(LogBuffer, ADR('0'));
		END_IF
		brsitoa(RtcGettime.hour, ADR(TmpStr));
		brsstrcat(LogBuffer, ADR(TmpStr));
		brsstrcat(LogBuffer, ADR(':'));
		IF(RtcGettime.minute < 10) THEN
			brsstrcat(LogBuffer, ADR('0'));
		END_IF
		brsitoa(RtcGettime.minute, ADR(TmpStr));
		brsstrcat(LogBuffer, ADR(TmpStr));
		brsstrcat(LogBuffer, ADR(':'));
		IF(RtcGettime.second < 10) THEN
			brsstrcat(LogBuffer, ADR('0'));
		END_IF
		brsitoa(RtcGettime.second, ADR(TmpStr));
		brsstrcat(LogBuffer, ADR(TmpStr));
		brsstrcat(LogBuffer, ADR('.'));
		IF(RtcGettime.millisec < 10) THEN
			brsstrcat(LogBuffer, ADR('00'));
		ELSIF(RtcGettime.millisec < 100) THEN
			brsstrcat(LogBuffer, ADR('0'));
		END_IF
		brsitoa(RtcGettime.millisec, ADR(TmpStr));
		brsstrcat(LogBuffer, ADR(TmpStr));
		// Add log message
		brsstrcat(LogBuffer, ADR(' '));
		brsstrcat(LogBuffer, ADR(LogMsg));
	END_IF
	LastMsg := LogMsg;

END_FUNCTION
```

#### revision.txt
```
Version 1.2
- Check remanent backup data against structure version to avoid data corruption

Version 1.1
- Handle division by zero
- Fix power off and power into the same shift days later does not trigger event
- Shift end event now uses power off date and time
- Fixed typos in function calls

Version 1.0

First public release
```

#### Common1.st - not listed in the package file held
```iecst
// -------------------------------------------------------------------------------------------
// Handle error state
FUNCTION CreateErrorState
	CreateLoggerEntry(exASSETINT_LOG_ERROR, ErrorMsg, ADR(Logger));

	StateError := State;
	State := exASSETINT_STATE_ERROR;

	DiagStatusID.ID := ErrorID;
	DiagStatusID.Code := UDINT_TO_UINT(StateError);
	DiagStatusID.Severity := Severity;

	CreateErrorState := ErrorID;
END_FUNCTION

// -------------------------------------------------------------------------------------------
// Handle log buffer
FUNCTION CreateLoggerEntry
	// Make sure we dont flood Logger
	IF LogMsg <> LastMsg AND LogLevel <= LOG_LEVEL THEN
		// Make sure log message fits
		IF brsstrlen(ADR(LogMsg)) > LOG_LEN THEN
			LogMsg := '*** log meassage exceeds maximum length ***';
		END_IF
		// Move ring buffer around
		brsmemmove(LogBuffer+LOG_LEN+1, LogBuffer, LOG_LEN*(LOG_NUM-1));
		brsstrcpy(LogBuffer, ADR(''));
		// Create time information
		RTC_gettime(ADR(RtcGettime));
		IF(RtcGettime.day < 10) THEN
			brsstrcat(LogBuffer, ADR('0'));
		END_IF
		brsitoa(RtcGettime.day, ADR(TmpStr));
		brsstrcat(LogBuffer, ADR(TmpStr));
		brsitoa(RtcGettime.day, ADR(TmpStr));
		brsstrcat(LogBuffer, ADR('.'));
		IF(RtcGettime.month < 10) THEN
			brsstrcat(LogBuffer, ADR('0'));
		END_IF
		brsitoa(RtcGettime.month, ADR(TmpStr));
		brsstrcat(LogBuffer, ADR(TmpStr));
		brsstrcat(LogBuffer, ADR(' '));
		IF(RtcGettime.hour < 10) THEN
			brsstrcat(LogBuffer, ADR('0'));
		END_IF
		brsitoa(RtcGettime.hour, ADR(TmpStr));
		brsstrcat(LogBuffer, ADR(TmpStr));
		brsstrcat(LogBuffer, ADR(':'));
		IF(RtcGettime.minute < 10) THEN
			brsstrcat(LogBuffer, ADR('0'));
		END_IF
		brsitoa(RtcGettime.minute, ADR(TmpStr));
		brsstrcat(LogBuffer, ADR(TmpStr));
		brsstrcat(LogBuffer, ADR(':'));
		IF(RtcGettime.second < 10) THEN
			brsstrcat(LogBuffer, ADR('0'));
		END_IF
		brsitoa(RtcGettime.second, ADR(TmpStr));
		brsstrcat(LogBuffer, ADR(TmpStr));
		brsstrcat(LogBuffer, ADR('.'));
		IF(RtcGettime.millisec < 10) THEN
			brsstrcat(LogBuffer, ADR('00'));
		ELSIF(RtcGettime.millisec < 100) THEN
			brsstrcat(LogBuffer, ADR('0'));
		END_IF
		brsitoa(RtcGettime.millisec, ADR(TmpStr));
		brsstrcat(LogBuffer, ADR(TmpStr));
		// Add log message
		brsstrcat(LogBuffer, ADR(' '));
		brsstrcat(LogBuffer, ADR(LogMsg));
	END_IF
	LastMsg := LogMsg;

END_FUNCTION
```

#### CreateDirStructure.st - not listed in the package file held
```iecst
// -------------------------------------------------------------------------------------------
// File version 1000
// -------------------------------------------------------------------------------------------
// Create folder structure
// -------------------------------------------------------------------------------------------
FUNCTION_BLOCK CreateDirStructure
	// -------------------------------------------------------------------------------------------
	// Reset everything when enable is false
	IF NOT Enable THEN
		Status := ERR_FUB_ENABLE_FALSE;
		State := 0;
	END_IF

	CASE State OF
		// -------------------------------------------------------------------------------------------
		// Wait for enable
		0:
			IF EDGEPOS(Enable) THEN
				DirCreate_0.enable := FALSE;
				DirCreate_0();

				DirCount := 0;
				TmpStr1 := CORE_FOLDER_NAME;
				brsstrcat(ADR(TmpStr1), ADR('0'));
				Status := ERR_FUB_BUSY;
				CreateLoggerEntry(exASSETINT_LOG_INFO, ADR('creating folder structure'), Logger);
				State := 1;
			END_IF

		// -------------------------------------------------------------------------------------------
		// Create folders
		1:
			DirCreate_0.enable := TRUE;
			DirCreate_0.pDevice := ADR(Device);
			DirCreate_0.pName := ADR(TmpStr1);
			DirCreate_0();

			// Folder created successful or folder already exsist
			IF DirCreate_0.status = ERR_OK OR DirCreate_0.status = fiERR_DIR_ALREADY_EXIST THEN
				// Generate log entry
				TmpStr2 := 'created folder ';
				brsstrcat(ADR(TmpStr2), ADR(TmpStr1));
				CreateLoggerEntry(exASSETINT_LOG_ALL, ADR(TmpStr2), Logger);

				// Create folders for 100 events each, finish when all folders are created
				DirCount := DirCount + 1;
				IF DirCount >= CORE_EVENT_NUM_MAX / CORE_EVENT_DIR_MAX THEN
					Status := ERR_OK;
					State := 0;

					// Generate next folder name
				ELSE
					TmpStr1 := CORE_FOLDER_NAME;
					brsitoa(DirCount, ADR(TmpStr2));
					brsstrcat(ADR(TmpStr1), ADR(TmpStr2));
				END_IF

				// Error
			ELSIF DirCreate_0.status <> ERR_FUB_BUSY THEN
				Status := DirCreate_0.status;
				State := 0;
			END_IF

	END_CASE;

END_FUNCTION_BLOCK
```

#### exAssetIntJobUI.st - not listed in the package file held
```iecst
// -------------------------------------------------------------------------------------------
// Job UI function block
FUNCTION_BLOCK exAssetIntJobListUI
	// -------------------------------------------------------------------------------------------
	// Reset everything when enable is false
	IF NOT Enable THEN
		StatusID := ERR_FUB_ENABLE_FALSE;
		Internal.State := exASSETINT_STATE_INIT_1;
		RETURN;
	END_IF

	CASE Internal.State OF

		// -------------------------------------------------------------------------------------------
		// Wait for enable
		exASSETINT_STATE_INIT_1:
			IF Enable THEN
				CreateLoggerEntry(exASSETINT_LOG_INFO, ADR('function block enabled'), Logger);

				// Make sure we have remanent buffer
				IF ADR(exLink) = 0 THEN
					// Set status, remember state, go to error state
					StatusID := CreateErrorState(ERR_ASSET_LINK, ADR('ERR: exLink is 0'), Logger, exCOM_SEV_ERROR, ADR(Internal.StateError), ADR(Internal.State), ADR(Info.Diag.StatusID));
					RETURN;
				END_IF
				// Make sure we have temporary buffer
				IF exLink.MemoryDb = 0 OR exLink.MemoryJob = 0 OR exLink.MemoryJob = 0 THEN
					// Set status, remember state, go to error state
					StatusID := CreateErrorState(ERR_ASSET_TEMP_MEMORY, ADR('ERR: no temp memory'), Logger, exCOM_SEV_ERROR, ADR(Internal.StateError), ADR(Internal.State), ADR(Info.Diag.StatusID));
					RETURN;
				END_IF
				// Make sure core function block is active
				IF NOT exLink.IsCoreActive THEN
					// Set status, remember state, go to error state
					StatusID := CreateErrorState(mpASSETINT_INF_WAIT_CORE_FB, ADR('ERR: core is not active'), Logger, exCOM_SEV_ERROR, ADR(Internal.StateError), ADR(Internal.State), ADR(Info.Diag.StatusID));
					RETURN;
				END_IF

				// Reset error and status
				Error := FALSE;
				StatusID := ERR_OK;
				Internal.SortingStartTimeOld := UDINT_TO_DINT(16#FFFFFFFF);

				Internal.State := exASSETINT_STATE_IDLE;
			END_IF

		// -------------------------------------------------------------------------------------------
		// Wait for new event
		exASSETINT_STATE_IDLE:
			// Reset record start when sorting direction changed
			IF UISetup.SortingStartTime <> Internal.SortingStartTimeOld THEN
				IF UISetup.SortingStartTime = exASSETINT_SORTING_ASC THEN
					Internal.RecordStart := 0;
				ELSE
					Internal.RecordStart := exLink.RecordCount;
				END_IF
			END_IF
			Internal.SortingStartTimeOld := UISetup.SortingStartTime;

			// Wait for core task to call update command
			IF exLink.RefreshJobUI AND exLink.RecordCount > 0 THEN
				CreateLoggerEntry(exASSETINT_LOG_INFO, ADR('refresh job data'), Logger);

				// Make correction for DESC sorting when record count changes
				IF UISetup.SortingStartTime = exASSETINT_SORTING_DESC AND Internal.RecordStart + exLink.RecordCount - Internal.RecordCountOld <= exLink.RecordCount THEN
					Internal.RecordStart := Internal.RecordStart + exLink.RecordCount - Internal.RecordCountOld;
				END_IF
				Internal.RecordCountOld := exLink.RecordCount;

				// Clear array and copy new data
				brsmemset(ADR(UIConnect.Output), 0, SIZEOF(UIConnect.Output));

				// Check how much data is left for ascending
				IF UISetup.SortingStartTime = exASSETINT_SORTING_ASC AND Internal.RecordStart + UI_JOB_LIST_IDX > exLink.RecordCount  THEN
					Internal.RecordNum := exLink.RecordCount - Internal.RecordStart - 1;
				// Check how much data is left for descending
				ELSIF UISetup.SortingStartTime = exASSETINT_SORTING_DESC AND Internal.RecordStart <= UI_JOB_LIST_IDX THEN
					Internal.RecordNum := Internal.RecordStart;
				ELSE
					Internal.RecordNum := UI_JOB_LIST_IDX;
				END_IF

				Internal.x := 0;
				REPEAT
					IF UISetup.SortingStartTime = exASSETINT_SORTING_ASC THEN
						brsmemcpy(ADR(Internal.RecordData), exLink.MemoryDb + (Internal.x + Internal.RecordStart)*SIZEOF(Internal.RecordData), SIZEOF(Internal.RecordData));
					ELSE
						brsmemcpy(ADR(Internal.RecordData), exLink.MemoryDb + (Internal.RecordStart - Internal.x - 1)*SIZEOF(Internal.RecordData), SIZEOF(Internal.RecordData));
					END_IF

					UIConnect.Output.JobStartTime[Internal.x] := Internal.RecordData.TimeStart;
					UIConnect.Output.JobEndTime[Internal.x] := Internal.RecordData.TimeEnd;
					UIConnect.Output.JobName[Internal.x] := Internal.RecordData.JobName;
					UIConnect.Output.CurrentUser[Internal.x] := Internal.RecordData.CurrentUser;
					UIConnect.Output.AdditionalData[Internal.x] := Internal.RecordData.AdditionalData;
					UIConnect.Output.TotalPieces[Internal.x] := Internal.RecordData.TotalPieces;
					UIConnect.Output.GoodPieces[Internal.x] := Internal.RecordData.GoodPieces;
					UIConnect.Output.RejectPieces[Internal.x] := Internal.RecordData.RejectPieces;
					UIConnect.Output.BadPieceRate[Internal.x] := Internal.RecordData.BadPieceRate;
					UIConnect.Output.TotalTime[Internal.x] := Internal.RecordData.TotalTime;
					UIConnect.Output.ScheduledDowntime[Internal.x] := Internal.RecordData.ScheduledDowntime;
					UIConnect.Output.UnscheduledDowntime[Internal.x] := Internal.RecordData.UnscheduledDowntime;
					UIConnect.Output.Uptime[Internal.x] := Internal.RecordData.Uptime;
					UIConnect.Output.GoodProductionTime[Internal.x] := Internal.RecordData.GoodProductionTime;
					UIConnect.Output.NominalProductionTime[Internal.x] := Internal.RecordData.NominalProductionTime;
					UIConnect.Output.NominalProductionRate[Internal.x] := Internal.RecordData.NominalProductionTimeRate;
					UIConnect.Output.UnscheduledDowntimeRate[Internal.x] := Internal.RecordData.UnscheduledDowntimeRate;
					UIConnect.Output.ProductionRate[Internal.x] := Internal.RecordData.CurrentProductionRate;
					UIConnect.Output.ShiftName[Internal.x] := Internal.RecordData.ShiftName;

					Internal.x := Internal.x + 1;

					UNTIL (Internal.x = Internal.RecordNum)
				END_REPEAT;

			END_IF
			exLink.RefreshJobUI := FALSE;

			// -------------------------------------------------------------------------------------------
			// Error state
		exASSETINT_STATE_ERROR:
			IF EDGEPOS(ErrorReset) THEN
				Internal.StateError := exASSETINT_STATE_NONE;
				Internal.State := exASSETINT_STATE_INIT_1;
			END_IF
	END_CASE;
END_FUNCTION_BLOCK
```

#### StoreEvent.st - not listed in the package file held
```iecst
// -------------------------------------------------------------------------------------------
// Create folder structure
// -------------------------------------------------------------------------------------------
FUNCTION_BLOCK StoreEvent
	// -------------------------------------------------------------------------------------------
	// Reset everything when enable is false
	IF NOT enable THEN
		status := ERR_FUB_ENABLE_FALSE;
		state := 0;
		RETURN;
	END_IF

	CASE state OF
		// -------------------------------------------------------------------------------------------
		// Wait for enable
		0:
			IF enable THEN
				// Reset function blocks
				FileOpen_0.enable := FALSE;
				FileOpen_0();
				FileCreate_0.enable := FALSE;
				FileCreate_0();
				FileWrite_0.enable := FALSE;
				FileWrite_0();
				FileClose_0.enable := FALSE;
				FileClose_0();

				// Generate file name
				tmpStr1 := 'events';
				brsitoa(record.ID/100, ADR(tmpStr2));
				brsstrcat(ADR(tmpStr1), ADR(tmpStr2));
				brsstrcat(ADR(tmpStr1), ADR('/event'));
				brsitoa(record.ID, ADR(tmpStr2));
				brsstrcat(ADR(tmpStr1), ADR(tmpStr2));

				status := ERR_FUB_BUSY;
				Logger(exASSETINT_LOG_INFO, 'creating new event', logger);
				state := state + 1;
			END_IF

		// -------------------------------------------------------------------------------------------
		// Open file
		1:
			FileOpen_0.enable := TRUE;
			FileOpen_0.pDevice := ADR(device);
			FileOpen_0.pFile := ADR(tmpStr1);
			FileOpen_0.mode := fiREAD_WRITE;
			FileOpen_0();

			// File opened successful
			IF FileOpen_0.status = ERR_OK THEN
				// Generate log entry
				tmpStr2 := 'opened event file ';
				brsstrcat(ADR(tmpStr2), ADR(tmpStr1));
				Logger(exASSETINT_LOG_ALL, tmpStr2, logger);

				// Remember ident go to next step
				ident := FileOpen_0.ident;
				state := 3;

			// Create event file when it does not exist
			ELSIF FileOpen_0.status = fiERR_FILE_NOT_FOUND  THEN
				state := 2;

			// Error
			ELSIF FileOpen_0.status <> ERR_FUB_BUSY THEN
				status := FileOpen_0.status;
				state := 0;
			END_IF

		// -------------------------------------------------------------------------------------------
		// Create file
		2:
			FileCreate_0.enable := TRUE;
			FileCreate_0.pDevice := ADR(device);
			FileCreate_0.pFile := ADR(tmpStr1);
			FileCreate_0();

			// File created successful
			IF FileCreate_0.status = ERR_OK THEN
				// Generate log entry
				tmpStr2 := 'created event file ';
				brsstrcat(ADR(tmpStr2), ADR(tmpStr1));
				Logger(exASSETINT_LOG_ALL, tmpStr2, logger);

				// Remember ident go to next step
				ident := FileCreate_0.ident;
				state := 3;

			// Error
			ELSIF FileCreate_0.status <> ERR_FUB_BUSY THEN
				status := FileCreate_0.status;
				state := 0;
			END_IF

		// -------------------------------------------------------------------------------------------
		// Write data
		3:
			FileWrite_0.enable := TRUE;
			FileWrite_0.ident := ident;
			FileWrite_0.pSrc := ADR(record);
			FileWrite_0.len := SIZEOF(record);
			FileWrite_0();

			// File created successful
			IF FileWrite_0.status = ERR_OK THEN
				// Generate log entry
				tmpStr2 := 'wrote event file ';
				brsstrcat(ADR(tmpStr2), ADR(tmpStr1));
				Logger(exASSETINT_LOG_ALL, tmpStr2, logger);

				// Go to next step
				state := 4;

			// Error
			ELSIF FileWrite_0.status <> ERR_FUB_BUSY THEN
				status := FileWrite_0.status;
				state := 0;
			END_IF

		// -------------------------------------------------------------------------------------------
		// Close file
		4:
			FileClose_0.enable := TRUE;
			FileClose_0.ident := ident;
			FileClose_0();

			// File created successful
			IF FileClose_0.status = ERR_OK THEN
				// Generate log entry
				tmpStr2 := 'closed event file ';
				brsstrcat(ADR(tmpStr2), ADR(tmpStr1));
				Logger(exASSETINT_LOG_ALL, tmpStr2, logger);

				// Finish up
				status := ERR_OK;
				state := 0;

			// Error
			ELSIF FileClose_0.status <> ERR_FUB_BUSY THEN
				status := FileWrite_0.status;
				state := 0;
			END_IF
	END_CASE;

END_FUNCTION_BLOCK
```

### Program Logical/exAssetInt/AssetTest

#### Variables.var
```iecst
VAR
	exAssetIntCore_0 : exAssetIntCore;
	exAssetIntPar : exAssetIntParType;
END_VAR
VAR RETAIN
	exBuffer : ARRAY[0..500] OF USINT;
END_VAR
```

#### Cyclic.st
```iecst
PROGRAM _CYCLIC
	exAssetIntCore_0.exLink := ADR(exBuffer);
	//exAssetIntCore_0.Enable := TRUE;
	exAssetIntCore_0.Parameters := ADR(exAssetIntPar);
	exAssetIntCore_0.DeviceName := ADR('ARsim');
	exAssetIntCore_0();

END_PROGRAM
```

#### Init.st
```iecst
PROGRAM _INIT
	exAssetIntPar.CurrentUser := 'TylerDurden';
	exAssetIntPar.Job := 'Cookies';
	exAssetIntPar.NominalProductionRate := 1000;

END_PROGRAM
```

- Visualisation Logical/Vis (not shown)

### Program Logical/Record

#### Variables.var
```iecst
VAR
	MpDataRecorder_0 : MpDataRecorder;
	CmdRecord : BOOL;
	MpDataRegPar_0 : MpDataRegPar;
	MpDataTableUI_0 : MpDataTableUI;
	gMpDataTableUIConnect : MpDataTableUIConnectType;
END_VAR
```

#### Cyclic.st
```iecst
PROGRAM _CYCLIC
    MpDataRecorder_0.MpLink := ADR(gDataRecorder);
    MpDataRecorder_0.Enable := TRUE;
    MpDataRecorder_0.Trigger := CmdRecord;
    MpDataRecorder_0.Record := MpDataRegPar_0.Active;
    MpDataRecorder_0();

    MpDataRegPar_0.MpLink := ADR(gDataRecorder);
    MpDataRegPar_0.Enable := MpDataRecorder_0.Active;
    MpDataRegPar_0.PVName := ADR('ShiftStatistics');
    MpDataRegPar_0.Description := ADR('xxx');
    MpDataRegPar_0.Unit := ADR('[°C]');
    MpDataRegPar_0();

//    MpDataTableUI_0.MpLink := ADR(gDataRecorder);
//    MpDataTableUI_0.Enable := MpDataRegPar_0.Active;
//    MpDataTableUI_0.UIConnect := ADR(gMpDataTableUIConnect);
//    MpDataTableUI_0();

END_PROGRAM
```

#### Exit.st
```iecst
PROGRAM _EXIT
    MpDataRecorder_0.Enable := FALSE;
    MpDataRecorder_0();
	MpDataRegPar_0.Enable := FALSE;
    MpDataRegPar_0();
//    MpDataTableUI_0.Enable := FALSE;
//    MpDataTableUI_0();
END_PROGRAM
```

#### Init.st
```iecst
PROGRAM _INIT
    MpDataRecorder_0.DeviceName := ADR('CFCard');
    MpDataRecorder_0.RecordMode := mpDATA_RECORD_MODE_TRIGGER;//mpDATA_RECORD_MODE_TIME;// mpDATA_RECORD_MODE_TRIGGER;
    MpDataRecorder_0.SamplingTime := T#2s; //T#60s;

END_PROGRAM
```

Listed in the project but not available here: Logical/Shift/Types.typ
